///////////////////////////////////////////////////////////////////////////////
// load values into akku1                                                    //
///////////////////////////////////////////////////////////////////////////////
      L    MB10;  // comment
// <- meta.block.fc.body meta.block.network
// ^^^^^^^^^^^^^^^^^^^^^^^^^ meta.block.fc.body meta.block.network
//    ^ keyword.operator.arithmetic.load
//         ^^^^ variable.language.address
//             ^ punctuation.terminator.statement
//                ^^ punctuation.definition.comment.begin
//                ^^^^^^^^^^ comment.line.double-slash
      L    MB[ LD0 ]; // comment
// <- meta.block.fc.body meta.block.network
// ^^^^^^^^^^^^^^^^^^^^^^^^^^^^ meta.block.fc.body meta.block.network
//         ^^^^^^^^^ meta.operand.numeric
//           ^^^^^^^ meta.brackets
//    ^ keyword.operator.arithmetic.load
//         ^^ variable.language.address
//           ^ punctuation.section.brackets.begin
//             ^^^ variable.language.address
//                 ^ punctuation.section.brackets.end
//                  ^ punctuation.terminator.statement
//                    ^^ punctuation.definition.comment.begin
//                    ^^^^^^^^^^ comment.line.double-slash
      L    MW10;  // comment
// <- meta.block.fc.body meta.block.network
// ^^^^^^^^^^^^^^^^^^^^^^^^^ meta.block.fc.body meta.block.network
//    ^ keyword.operator.arithmetic.load
//         ^^^^ variable.language.address
//             ^ punctuation.terminator.statement
//                ^^ punctuation.definition.comment.begin
//                ^^^^^^^^^^ comment.line.double-slash
      L    MW[ LD0 ]; // comment
// <- meta.block.fc.body meta.block.network
// ^^^^^^^^^^^^^^^^^^^^^^^^^^^^ meta.block.fc.body meta.block.network
//         ^^^^^^^^^ meta.operand.numeric
//           ^^^^^^^ meta.brackets
//    ^ keyword.operator.arithmetic.load
//         ^^ variable.language.address
//           ^ punctuation.section.brackets.begin
//             ^^^ variable.language.address
//                 ^ punctuation.section.brackets.end
//                  ^ punctuation.terminator.statement
//                    ^^ punctuation.definition.comment.begin
//                    ^^^^^^^^^^ comment.line.double-slash
      L    MD10;  // comment
// <- meta.block.fc.body meta.block.network
// ^^^^^^^^^^^^^^^^^^^^^^^^^ meta.block.fc.body meta.block.network
//    ^ keyword.operator.arithmetic.load
//         ^^^^ variable.language.address
//             ^ punctuation.terminator.statement
//                ^^ punctuation.definition.comment.begin
//                ^^^^^^^^^^ comment.line.double-slash
      L    MD[ LD0 ]; // comment
// <- meta.block.fc.body meta.block.network
// ^^^^^^^^^^^^^^^^^^^^^^^^^^^^ meta.block.fc.body meta.block.network
//         ^^^^^^^^^ meta.operand.numeric
//           ^^^^^^^ meta.brackets
//    ^ keyword.operator.arithmetic.load
//         ^^ variable.language.address
//           ^ punctuation.section.brackets.begin
//             ^^^ variable.language.address
//                 ^ punctuation.section.brackets.end
//                  ^ punctuation.terminator.statement
//                    ^^ punctuation.definition.comment.begin
//                    ^^^^^^^^^^ comment.line.double-slash
      L    M10.0;  // comment
// <- meta.block.fc.body meta.block.network
// ^^^^^^^^^^^^^^^^^^^^^^^^^^ meta.block.fc.body meta.block.network
//    ^ keyword.operator.arithmetic.load
//         ^^^^^ invalid.illegal
//              ^ punctuation.terminator.statement
//                 ^^ punctuation.definition.comment.begin
//                 ^^^^^^^^^^ comment.line.double-slash
      L    LB10;  // comment
// <- meta.block.fc.body meta.block.network
// ^^^^^^^^^^^^^^^^^^^^^^^^^ meta.block.fc.body meta.block.network
//    ^ keyword.operator.arithmetic.load
//         ^^^^ variable.language.address
//             ^ punctuation.terminator.statement
//                ^^ punctuation.definition.comment.begin
//                ^^^^^^^^^^ comment.line.double-slash
      L    LB[ LD0 ]; // comment
// <- meta.block.fc.body meta.block.network
// ^^^^^^^^^^^^^^^^^^^^^^^^^^^^ meta.block.fc.body meta.block.network
//         ^^^^^^^^^ meta.operand.numeric
//           ^^^^^^^ meta.brackets
//    ^ keyword.operator.arithmetic.load
//         ^^ variable.language.address
//           ^ punctuation.section.brackets.begin
//             ^^^ variable.language.address
//                 ^ punctuation.section.brackets.end
//                  ^ punctuation.terminator.statement
//                    ^^ punctuation.definition.comment.begin
//                    ^^^^^^^^^^ comment.line.double-slash
      L    LW10;  // comment
// <- meta.block.fc.body meta.block.network
// ^^^^^^^^^^^^^^^^^^^^^^^^^ meta.block.fc.body meta.block.network
//    ^ keyword.operator.arithmetic.load
//         ^^^^ variable.language.address
//             ^ punctuation.terminator.statement
//                ^^ punctuation.definition.comment.begin
//                ^^^^^^^^^^ comment.line.double-slash
      L    LW[ LD0 ]; // comment
// <- meta.block.fc.body meta.block.network
// ^^^^^^^^^^^^^^^^^^^^^^^^^^^^ meta.block.fc.body meta.block.network
//         ^^^^^^^^^ meta.operand.numeric
//           ^^^^^^^ meta.brackets
//    ^ keyword.operator.arithmetic.load
//         ^^ variable.language.address
//           ^ punctuation.section.brackets.begin
//             ^^^ variable.language.address
//                 ^ punctuation.section.brackets.end
//                  ^ punctuation.terminator.statement
//                    ^^ punctuation.definition.comment.begin
//                    ^^^^^^^^^^ comment.line.double-slash
      L    LD10;  // comment
// <- meta.block.fc.body meta.block.network
// ^^^^^^^^^^^^^^^^^^^^^^^^^ meta.block.fc.body meta.block.network
//    ^ keyword.operator.arithmetic.load
//         ^^^^ variable.language.address
//             ^ punctuation.terminator.statement
//                ^^ punctuation.definition.comment.begin
//                ^^^^^^^^^^ comment.line.double-slash
      L    LD[ LD0 ]; // comment
// <- meta.block.fc.body meta.block.network
// ^^^^^^^^^^^^^^^^^^^^^^^^^^^^ meta.block.fc.body meta.block.network
//         ^^^^^^^^^ meta.operand.numeric
//           ^^^^^^^ meta.brackets
//    ^ keyword.operator.arithmetic.load
//         ^^ variable.language.address
//           ^ punctuation.section.brackets.begin
//             ^^^ variable.language.address
//                 ^ punctuation.section.brackets.end
//                  ^ punctuation.terminator.statement
//                    ^^ punctuation.definition.comment.begin
//                    ^^^^^^^^^^ comment.line.double-slash
      L    L10.0;  // comment
// <- meta.block.fc.body meta.block.network
// ^^^^^^^^^^^^^^^^^^^^^^^^^^ meta.block.fc.body meta.block.network
//    ^ keyword.operator.arithmetic.load
//         ^^^^^ invalid.illegal
//              ^ punctuation.terminator.statement
//                 ^^ punctuation.definition.comment.begin
//                 ^^^^^^^^^^ comment.line.double-slash
      L     T 10;  // comment
// <- meta.block.fc.body meta.block.network
// ^^^^^^^^^^^^^^^^^^^^^^^^^^ meta.block.fc.body meta.block.network
//    ^ keyword.operator.arithmetic.load
//          ^^^^ variable.language.timer
//              ^ punctuation.terminator.statement
//                 ^^ punctuation.definition.comment.begin
//                 ^^^^^^^^^^ comment.line.double-slash
      L     T [MW10];  // comment
// <- meta.block.fc.body meta.block.network
// ^^^^^^^^^^^^^^^^^^^^^^^^^^^^^ meta.block.fc.body meta.block.network
//     ^^^^^ meta.operand.numeric - meta.address
//          ^^ meta.operand.numeric meta.address.indirect - meta.brackets
//            ^^^^^^ meta.address.indirect meta.brackets
//                  ^^^^^^^^^^^^^^ - meta.operand
//    ^ keyword.operator.arithmetic.load
//          ^ variable.language.timer
//            ^ punctuation.section.brackets.begin
//             ^^^^ variable.language.address
//                 ^ punctuation.section.brackets.end
//                  ^ punctuation.terminator.statement
//                     ^^ punctuation.definition.comment.begin
//                     ^^^^^^^^^^ comment.line.double-slash
      L     Z 10;  // comment
// <- meta.block.fc.body meta.block.network
// ^^^^^^^^^^^^^^^^^^^^^^^^^^ meta.block.fc.body meta.block.network
//    ^ keyword.operator.arithmetic.load
//          ^^^^ variable.language.counter
//              ^ punctuation.terminator.statement
//                 ^^ punctuation.definition.comment.begin
//                 ^^^^^^^^^^ comment.line.double-slash
      L     Z [MW10];  // comment
// <- meta.block.fc.body meta.block.network
// ^^^^^^^^^^^^^^^^^^^^^^^^^^^^^ meta.block.fc.body meta.block.network
//     ^^^^^ meta.operand.numeric - meta.address
//          ^^ meta.operand.numeric meta.address.indirect - meta.brackets
//            ^^^^^^ meta.address.indirect meta.brackets
//                  ^^^^^^^^^^^^^^ - meta.operand
//    ^ keyword.operator.arithmetic.load
//          ^ variable.language.counter
//            ^ punctuation.section.brackets.begin
//             ^^^^ variable.language.address
//                 ^ punctuation.section.brackets.end
//                  ^ punctuation.terminator.statement
//                     ^^ punctuation.definition.comment.begin
//                     ^^^^^^^^^^ comment.line.double-slash
      L     DBNO;  // comment
// <- meta.block.fc.body meta.block.network
// ^^^^^^^^^^^^^^^^^^^^^^^^^^ meta.block.fc.body meta.block.network
//    ^ keyword.operator.arithmetic.load
//          ^^^^ variable.language
//              ^ punctuation.terminator.statement
//                 ^^ punctuation.definition.comment.begin
//                 ^^^^^^^^^^ comment.line.double-slash
      L     DINO;  // comment
// <- meta.block.fc.body meta.block.network
// ^^^^^^^^^^^^^^^^^^^^^^^^^^ meta.block.fc.body meta.block.network
//    ^ keyword.operator.arithmetic.load
//          ^^^^ variable.language
//              ^ punctuation.terminator.statement
//                 ^^ punctuation.definition.comment.begin
//                 ^^^^^^^^^^ comment.line.double-slash
      L     DBB  140;  // comment
// <- meta.block.fc.body meta.block.network
// ^^^^^^^^^^^^^^^^^^^^^^^^^^^^^^ meta.block.fc.body meta.block.network
//    ^ keyword.operator.arithmetic.load
//          ^^^^^^^^ variable.language.address
//                  ^ punctuation.terminator.statement
//                     ^^ punctuation.definition.comment.begin
//                     ^^^^^^^^^^ comment.line.double-slash
      L     DBW  140;  // comment
// <- meta.block.fc.body meta.block.network
// ^^^^^^^^^^^^^^^^^^^^^^^^^^^^^^ meta.block.fc.body meta.block.network
//    ^ keyword.operator.arithmetic.load
//          ^^^^^^^^ variable.language.address
//                  ^ punctuation.terminator.statement
//                     ^^ punctuation.definition.comment.begin
//                     ^^^^^^^^^^ comment.line.double-slash
      L     DBD  140;  // comment
// <- meta.block.fc.body meta.block.network
// ^^^^^^^^^^^^^^^^^^^^^^^^^^^^^^ meta.block.fc.body meta.block.network
//    ^ keyword.operator.arithmetic.load
//          ^^^^^^^^ variable.language.address
//                  ^ punctuation.terminator.statement
//                     ^^ punctuation.definition.comment.begin
//                     ^^^^^^^^^^ comment.line.double-slash
      L     DIB  140;  // comment
// <- meta.block.fc.body meta.block.network
// ^^^^^^^^^^^^^^^^^^^^^^^^^^^^^^ meta.block.fc.body meta.block.network
//    ^ keyword.operator.arithmetic.load
//          ^^^^^^^^ variable.language.address
//                  ^ punctuation.terminator.statement
//                     ^^ punctuation.definition.comment.begin
//                     ^^^^^^^^^^ comment.line.double-slash
      L     DIW  140;  // comment
// <- meta.block.fc.body meta.block.network
// ^^^^^^^^^^^^^^^^^^^^^^^^^^^^^^ meta.block.fc.body meta.block.network
//    ^ keyword.operator.arithmetic.load
//          ^^^^^^^^ variable.language.address
//                  ^ punctuation.terminator.statement
//                     ^^ punctuation.definition.comment.begin
//                     ^^^^^^^^^^ comment.line.double-slash
      L     DID  140;  // comment
// <- meta.block.fc.body meta.block.network
// ^^^^^^^^^^^^^^^^^^^^^^^^^^^^^^ meta.block.fc.body meta.block.network
//    ^ keyword.operator.arithmetic.load
//          ^^^^^^^^ variable.language.address
//                  ^ punctuation.terminator.statement
//                     ^^ punctuation.definition.comment.begin
//                     ^^^^^^^^^^ comment.line.double-slash
      L    DB200.DBB20;  // comment
// <- meta.block.fc.body meta.block.network
// ^^^^^^^^^^^^^^^^^^^^^^^^^^^^^^^^ meta.block.fc.body meta.block.network
//    ^ keyword.operator.arithmetic.load
//         ^^^^^ variable.language.db
//              ^ punctuation.accessor.dot
//               ^^^^^ variable.language.address
//                    ^ punctuation.terminator.statement
//                       ^^ punctuation.definition.comment.begin
//                       ^^^^^^^^^^ comment.line.double-slash
      L    DB200.DBW20;  // comment
// <- meta.block.fc.body meta.block.network
// ^^^^^^^^^^^^^^^^^^^^^^^^^^^^^^^^ meta.block.fc.body meta.block.network
//    ^ keyword.operator.arithmetic.load
//         ^^^^^ variable.language.db
//              ^ punctuation.accessor.dot
//               ^^^^^ variable.language.address
//                    ^ punctuation.terminator.statement
//                       ^^ punctuation.definition.comment.begin
//                       ^^^^^^^^^^ comment.line.double-slash
      L    DB200.DBD20;  // comment
// <- meta.block.fc.body meta.block.network
// ^^^^^^^^^^^^^^^^^^^^^^^^^^^^^^^^ meta.block.fc.body meta.block.network
//    ^ keyword.operator.arithmetic.load
//         ^^^^^ variable.language.db
//              ^ punctuation.accessor.dot
//               ^^^^^ variable.language.address
//                    ^ punctuation.terminator.statement
//                       ^^ punctuation.definition.comment.begin
//                       ^^^^^^^^^^ comment.line.double-slash
      L    DB200.DBX20.0;  // comment
// <- meta.block.fc.body meta.block.network
// ^^^^^^^^^^^^^^^^^^^^^^^^^^^^^^^^^^ meta.block.fc.body meta.block.network
//    ^ keyword.operator.arithmetic.load
//         ^^^^^^^^^^^^^ invalid.illegal
//                      ^ punctuation.terminator.statement
//                         ^^ punctuation.definition.comment.begin
//                         ^^^^^^^^^^ comment.line.double-slash
      L    "datablock".struct[ 4 ].value;  // comment
// <- meta.block.fc.body meta.block.network
// ^^^^^^^^^^^^^^^^^^^^^^^^^^^^^^^^^^^^^^^^^^^^^ meta.block.fc.body meta.block.network
//         ^^^^^^^^^^^^^^^^^^^^^^^^^^^^^ meta.path
//    ^ keyword.operator.arithmetic.load
//         ^ punctuation.definition.variable.begin
//         ^^^^^^^^^^^ variable.namespace
//                   ^ punctuation.definition.variable.end
//                    ^ punctuation.accessor.dot
//                     ^^^^^^ variable.namespace
//                           ^ punctuation.section.brackets.begin
//                           ^^^^^ meta.brackets
//                             ^ meta.number.integer constant.numeric.value
//                               ^ punctuation.section.brackets.end
//                                ^ punctuation.accessor.dot
//                                 ^^^^^ variable.other.member
//                                      ^ punctuation.terminator.statement
//                                         ^^ punctuation.definition.comment.begin
//                                         ^^^^^^^^^^ comment.line.double-slash
      L    "datablock".struct.value;  // comment
// <- meta.block.fc.body meta.block.network
// ^^^^^^^^^^^^^^^^^^^^^^^^^^^^^^^^^^^^^^^^^^^^^ meta.block.fc.body meta.block.network
//         ^^^^^^^^^^^^^^^^^^^^^^^^ meta.path
//    ^ keyword.operator.arithmetic.load
//         ^ punctuation.definition.variable.begin
//         ^^^^^^^^^^^ variable.namespace
//                   ^ punctuation.definition.variable.end
//                    ^ punctuation.accessor.dot
//                     ^^^^^^ variable.namespace
//                           ^ punctuation.accessor.dot
//                            ^^^^^ variable.other.member
//                                 ^ punctuation.terminator.statement
//                                    ^^ punctuation.definition.comment.begin
//                                    ^^^^^^^^^^ comment.line.double-slash
      L    #local[1].array[0].value[ 10 ];  // comment
// <- meta.block.fc.body meta.block.network
// ^^^^^^^^^^^^^^^^^^^^^^^^^^^^^^^^^^^^^^^^^^^^^^ meta.block.fc.body meta.block.network
//    ^ keyword.operator.arithmetic.load
//         ^ punctuation.definition.variable
//         ^^^^^^ variable.namespace
//               ^ punctuation.section.brackets.begin
//               ^^^ meta.brackets
//                ^ meta.number.integer constant.numeric.value
//                 ^ punctuation.section.brackets.end
//                  ^ punctuation.accessor.dot
//                   ^^^^^ variable.namespace
//                        ^ punctuation.section.brackets.begin
//                        ^^^ meta.brackets
//                         ^ meta.number.integer constant.numeric.value
//                          ^ punctuation.section.brackets.end
//                           ^ punctuation.accessor.dot
//                            ^^^^^ variable.other.member
//                                 ^ punctuation.section.brackets.begin
//                                 ^^^^^^ meta.brackets
//                                   ^^ meta.number.integer constant.numeric.value
//                                      ^ punctuation.section.brackets.end
//                                       ^ punctuation.terminator.statement
//                                          ^^ punctuation.definition.comment.begin
//                                          ^^^^^^^^^^ comment.line.double-slash
      L    myNamedValueType#value; // TIA only
//^^^^^^^^^^^^^^^^^^^^^^^^^^^^^^^^ meta.block.fc.body.plc meta.block.network.plc
//    ^ keyword.operator.arithmetic.load.plc
//     ^^^^^^^^^^^^^^^^^^^^^^^^^^ meta.operand.numeric.plc
//         ^^^^^^^^^^^^^^^^ storage.type.enum.plc
//                         ^ punctuation.accessor.plc
//                          ^^^^^ constant.other.enum.plc
//                               ^ punctuation.terminator.statement.plc
      L    "Fancy Named Value Type"#"fancy value"; // TIA only
//^^^^^^^^^^^^^^^^^^^^^^^^^^^^^^^^^^^^^^^^^^^^^^^^ meta.block.fc.body.plc meta.block.network.plc
//    ^ keyword.operator.arithmetic.load.plc
//     ^^^^^^^^^^^^^^^^^^^^^^^^^^^^^^^^^^^^^^^^^^ meta.operand.numeric.plc
//         ^^^^^^^^^^^^^^^^^^^^^^^^ storage.type.enum.plc
//         ^ punctuation.definition.constant.begin.plc
//                                ^ punctuation.definition.constant.end.plc
//                                 ^ punctuation.accessor.plc
//                                  ^^^^^^^^^^^^^ constant.other.enum.plc
//                                  ^ punctuation.definition.constant.begin.plc
//                                              ^ punctuation.definition.constant.end.plc
//                                               ^ punctuation.terminator.statement.plc
      L    P# P0.0; // comment
// <- meta.block.fc.body meta.block.network
// ^^^^^^^^^^^^^^^^^^^^^^^^^^^^^ meta.block.fc.body meta.block.network
//    ^ keyword.operator.arithmetic.load
//         ^^^^^^^ constant.language.pointer
//         ^ storage.type.pointer
//          ^ punctuation.separator.type
//              ^ punctuation.separator.decimal
//                ^ punctuation.terminator.statement
//                  ^^ punctuation.definition.comment.begin
//                  ^^^^^^^^^^ comment.line.double-slash
      L    P##local;  // comment
// <- meta.block.fc.body meta.block.network
// ^^^^^^^^^^^^^^^^^^^^^^^^^^^^^ meta.block.fc.body meta.block.network
//    ^ keyword.operator.arithmetic.load
//         ^ storage.type.pointer
//          ^ punctuation.separator.type
//           ^ punctuation.definition.variable
//            ^^^^^ variable.other.local
//                 ^ punctuation.terminator.statement
//                    ^^ punctuation.definition.comment.begin
//                    ^^^^^^^^^^ comment.line.double-slash
      L    P#120.4;  // comment
// <- meta.block.fc.body meta.block.network
// ^^^^^^^^^^^^^^^^^^^^^^^^^^^^^ meta.block.fc.body meta.block.network
//    ^ keyword.operator.arithmetic.load
//         ^^^^^^^ constant.language.pointer
//         ^ storage.type.pointer
//          ^ punctuation.separator.type
//                ^ punctuation.terminator.statement
//                   ^^ punctuation.definition.comment.begin
//                   ^^^^^^^^^^ comment.line.double-slash
      L    P#DBX120.4;  // comment
// <- meta.block.fc.body meta.block.network
// ^^^^^^^^^^^^^^^^^^^^^^^^^^^^^^^ meta.block.fc.body meta.block.network
//    ^ keyword.operator.arithmetic.load
//         ^^^^^^^^^^ constant.language.pointer
//         ^ storage.type.pointer
//          ^ punctuation.separator.type
//                 ^ punctuation.separator.decimal
//                   ^ punctuation.terminator.statement
//                      ^^ punctuation.definition.comment.begin
//                      ^^^^^^^^^^ comment.line.double-slash
      L    P#DB2.DBX120.4;  // comment
// <- meta.block.fc.body meta.block.network
// ^^^^^^^^^^^^^^^^^^^^^^^^^^^^^^^^^^^^ meta.block.fc.body meta.block.network
//    ^ keyword.operator.arithmetic.load
//         ^^^^^^^^^^^^^^ constant.language.pointer
//         ^ storage.type.pointer
//          ^ punctuation.separator.type
//              ^ punctuation.accessor.dot
//                     ^ punctuation.separator.decimal
//                       ^ punctuation.terminator.statement
//                          ^^ punctuation.definition.comment.begin
//                          ^^^^^^^^^^ comment.line.double-slash
      L    2#0000_0000_0000_0000_0000_0000_0000_0000 ;
// <- meta.block.fc.body meta.block.network
// ^^^^^^^^^^^^^^^^^^^^^^^^^^^^^^^^^^^^^^^^^^^^^^^^^^^^ meta.block.fc.body meta.block.network
//    ^ keyword.operator.arithmetic.load
//         ^^^^^^^^^^^^^^^^^^^^^^^^^^^^^^^^^^^^^^^^^ meta.number.integer.binary
//         ^ constant.numeric.base - punctuation
//          ^ constant.numeric.base punctuation.separator.base
//           ^^^^^^^^^^^^^^^^^^^^^^^^^^^^^^^^^^^^^^^ constant.numeric.value
//               ^ punctuation.separator.digits
//                    ^ punctuation.separator.digits
//                         ^ punctuation.separator.digits
//                              ^ punctuation.separator.digits
//                                   ^ punctuation.separator.digits
//                                        ^ punctuation.separator.digits
//                                             ^ punctuation.separator.digits
//                                                  ^ - invalid
//                                                   ^ punctuation.terminator.statement
//                                                    ^ - invalid
      L    2#1111_1111_1111_1111_1111_1111_1111_1111 ;
// <- meta.block.fc.body meta.block.network
// <- meta.block.fc.body meta.block.network
// ^^^^^^^^^^^^^^^^^^^^^^^^^^^^^^^^^^^^^^^^^^^^^^^^^^^^ meta.block.fc.body meta.block.network
//    ^ keyword.operator.arithmetic.load
//         ^^^^^^^^^^^^^^^^^^^^^^^^^^^^^^^^^^^^^^^^^ meta.number.integer.binary
//         ^ constant.numeric.base - punctuation
//          ^ constant.numeric.base punctuation.separator.base
//           ^^^^^^^^^^^^^^^^^^^^^^^^^^^^^^^^^^^^^^^ constant.numeric.value
//               ^ punctuation.separator.digits
//                    ^ punctuation.separator.digits
//                         ^ punctuation.separator.digits
//                              ^ punctuation.separator.digits
//                                   ^ punctuation.separator.digits
//                                        ^ punctuation.separator.digits
//                                             ^ punctuation.separator.digits
//                                                  ^ - invalid
//                                                   ^ punctuation.terminator.statement
//                                                    ^ - invalid
      L    2#1121_1111_1A11_1111_111_11011_1111_1111 ;
// <- meta.block.fc.body meta.block.network
// ^^^^^^^^^^^^^^^^^^^^^^^^^^^^^^^^^^^^^^^^^^^^^^^^^^^^ meta.block.fc.body meta.block.network
//    ^ keyword.operator.arithmetic.load
//         ^^^^^^^^^^^^^^^^^^^^^^^^^^^^^^^^^^^^^^^^^ meta.number.integer.binary
//         ^ constant.numeric.base - punctuation
//          ^ constant.numeric.base punctuation.separator.base
//           ^^^^^^^^^^^^^^^^^^^^^^^^^^^^^^^^^^^^^^^ constant.numeric.value
//             ^ invalid.illegal.digits
//               ^ punctuation.separator.digits
//                    ^ punctuation.separator.digits
//                      ^ invalid.illegal.digits
//                         ^ punctuation.separator.digits
//                              ^ punctuation.separator.digits
//                                  ^ punctuation.separator.digits
//                                        ^ punctuation.separator.digits
//                                             ^ punctuation.separator.digits
//                                                  ^ - invalid
//                                                   ^ punctuation.terminator.statement
//                                                    ^ - invalid
      L    B#16#0 ;
// <- meta.block.fc.body meta.block.network
// ^^^^^^^^^^^^^^^^^ meta.block.fc.body meta.block.network
//    ^ keyword.operator.arithmetic.load
//         ^^^^^^ meta.number.integer.hexadecimal
//         ^ storage.type.integer
//          ^ punctuation.separator.type
//           ^^ constant.numeric.base - punctuation
//             ^ constant.numeric.base punctuation.separator.base
//              ^ constant.numeric.value
//               ^ - invalid
//                ^ punctuation.terminator.statement
//                 ^ - invalid
      L    byte#16#0 ;
// <- meta.block.fc.body meta.block.network
// ^^^^^^^^^^^^^^^^^^^^ meta.block.fc.body meta.block.network
//    ^ keyword.operator.arithmetic.load
//         ^^^^^^^^^ meta.number.integer.hexadecimal
//         ^^^^ storage.type.integer
//             ^ punctuation.separator.type
//              ^^ constant.numeric.base - punctuation
//                ^ constant.numeric.base punctuation.separator.base
//                 ^ constant.numeric.value
//                  ^ - invalid
//                   ^ punctuation.terminator.statement
//                    ^ - invalid
      L    W#16#0 ;
// <- meta.block.fc.body meta.block.network
// ^^^^^^^^^^^^^^^^^ meta.block.fc.body meta.block.network
//    ^ keyword.operator.arithmetic.load
//         ^^^^^^ meta.number.integer.hexadecimal
//         ^ storage.type.integer
//          ^ punctuation.separator.type
//           ^^ constant.numeric.base - punctuation
//             ^ constant.numeric.base punctuation.separator.base
//              ^ constant.numeric.value
//               ^ - invalid
//                ^ punctuation.terminator.statement
//                 ^ - invalid
      L    word#16#0 ;
// <- meta.block.fc.body meta.block.network
// ^^^^^^^^^^^^^^^^^^^^ meta.block.fc.body meta.block.network
//    ^ keyword.operator.arithmetic.load
//         ^^^^^^^^^ meta.number.integer.hexadecimal
//         ^^^^ storage.type.integer
//             ^ punctuation.separator.type
//              ^^ constant.numeric.base - punctuation
//                ^ constant.numeric.base punctuation.separator.base
//                 ^ constant.numeric.value
//                  ^ - invalid
//                   ^ punctuation.terminator.statement
//                    ^ - invalid
      L    DW#16#0 ;
// <- meta.block.fc.body meta.block.network
// ^^^^^^^^^^^^^^^^^ meta.block.fc.body meta.block.network
//    ^ keyword.operator.arithmetic.load
//         ^^^^^^^ meta.number.integer.hexadecimal
//         ^^ storage.type.integer
//           ^ punctuation.separator.type
//            ^^ constant.numeric.base - punctuation
//              ^ constant.numeric.base punctuation.separator.base
//               ^ constant.numeric.value
//                ^ - invalid
//                 ^ punctuation.terminator.statement
//                  ^ - invalid
      L    dword#16#0 ;
// <- meta.block.fc.body meta.block.network
// ^^^^^^^^^^^^^^^^^^^^^ meta.block.fc.body meta.block.network
//    ^ keyword.operator.arithmetic.load
//         ^^^^^^^^^ meta.number.integer.hexadecimal
//         ^^^^^ storage.type.integer
//              ^ punctuation.separator.type
//               ^^ constant.numeric.base - punctuation
//                 ^ constant.numeric.base punctuation.separator.base
//                  ^ constant.numeric.value
//                   ^ - invalid
//                    ^ punctuation.terminator.statement
//                     ^ - invalid
      L    16 ;
// <- meta.block.fc.body meta.block.network
// ^^^^^^^^^^^^^^^ meta.block.fc.body meta.block.network
//    ^ keyword.operator.arithmetic.load
//         ^^ meta.number.integer.decimal
//         ^^ constant.numeric.value
//           ^ - invalid
//            ^ punctuation.terminator.statement
//             ^ - invalid
      L    -16 ;
// <- meta.block.fc.body meta.block.network
// ^^^^^^^^^^^^^^^ meta.block.fc.body meta.block.network
//    ^ keyword.operator.arithmetic.load
//         ^^^ meta.number.integer.decimal
//         ^ keyword.operator.arithmetic - constant.numeric.value
//          ^^ constant.numeric.value - keyword.operator
//            ^ - invalid
//             ^ punctuation.terminator.statement
//              ^ - invalid
      L    L#16 ;
// <- meta.block.fc.body meta.block.network
// ^^^^^^^^^^^^^^^ meta.block.fc.body meta.block.network
//    ^ keyword.operator.arithmetic.load
//         ^^^^ meta.number.integer.decimal
//         ^ storage.type.integer
//          ^ punctuation.separator.type
//           ^^ constant.numeric.value
//             ^ - invalid
//              ^ punctuation.terminator.statement
//               ^ - invalid
      L    L#-16 ;
// <- meta.block.fc.body meta.block.network
// ^^^^^^^^^^^^^^^ meta.block.fc.body meta.block.network
//    ^ keyword.operator.arithmetic.load
//         ^^^^^ meta.number.integer.decimal
//         ^ storage.type.integer
//          ^ punctuation.separator.type
//           ^ keyword.operator.arithmetic - constant.numeric.value
//            ^^ constant.numeric.value - keyword.operator
//              ^ - invalid
//               ^ punctuation.terminator.statement
//                ^ - invalid
      L    2.0323e+002 ;
// <- meta.block.fc.body meta.block.network
// ^^^^^^^^^^^^^^^^^^^^^^ meta.block.fc.body meta.block.network
//    ^ keyword.operator.arithmetic.load
//         ^^^^^^^^^^^ meta.number.float.decimal constant.numeric.value
//          ^ punctuation.separator.decimal
//                    ^ - invalid
//                     ^ punctuation.terminator.statement
//                      ^ - invalid
      L    -2.0323e-002 ;
// <- meta.block.fc.body meta.block.network
// ^^^^^^^^^^^^^^^^^^^^^^ meta.block.fc.body meta.block.network
//    ^ keyword.operator.arithmetic.load
//         ^^^^^^^^^^^ meta.number.float.decimal
//         ^ keyword.operator.arithmetic - constant.numeric.value
//          ^^^^^^^^^^^ constant.numeric.value - keyword.operator
//           ^ punctuation.separator.decimal
//                     ^ - invalid
//                      ^ punctuation.terminator.statement
//                       ^ - invalid
      L    C#200 ;
// <- meta.block.fc.body meta.block.network
// ^^^^^^^^^^^^^^^^ meta.block.fc.body meta.block.network
//    ^ keyword.operator.arithmetic.load
//         ^^^^^ meta.number.counter.s5
//         ^ storage.type.counter
//          ^ punctuation.separator.type
//           ^^^ constant.numeric.value
//              ^ - invalid
//               ^ punctuation.terminator.statement
//                ^ - invalid
      L     S5T#50MS ;
// <- meta.block.fc.body meta.block.network
// ^^^^^^^^^^^^^^^^^^^ meta.block.fc.body meta.block.network
//    ^ keyword.operator.arithmetic.load
//          ^^^^^^^^ meta.number.time.s5
//          ^^^ storage.type.time
//             ^ punctuation.separator.type
//              ^^ constant.numeric.value.millisecond
//                ^^ constant.numeric.suffix
//                  ^ - invalid
//                   ^ punctuation.terminator.statement
//                    ^ - invalid
      L     S5T#50S ;
// <- meta.block.fc.body meta.block.network
// ^^^^^^^^^^^^^^^^^^ meta.block.fc.body meta.block.network
//    ^ keyword.operator.arithmetic.load
//          ^^^^^^^ meta.number.time.s5
//          ^^^ storage.type.time
//             ^ punctuation.separator.type
//              ^^ constant.numeric.value.second
//                ^ constant.numeric.suffix
//                 ^ - invalid
//                  ^ punctuation.terminator.statement
//                   ^ - invalid
      L     S5T#50M ; //Lade 3000s Sekunden
// <- meta.block.fc.body meta.block.network
// ^^^^^^^^^^^^^^^^^^ meta.block.fc.body meta.block.network
//    ^ keyword.operator.arithmetic.load
//          ^^^^^^^ meta.number.time.s5
//          ^^^ storage.type.time
//             ^ punctuation.separator.type
//              ^^ constant.numeric.value.minute
//                ^ constant.numeric.suffix
//                 ^ - invalid
//                  ^ punctuation.terminator.statement
//                   ^ - invalid
//                    ^^^^^^^^^^^^^^^^^^^^^ comment.line
      L     S5T#1H ;
// <- meta.block.fc.body meta.block.network
// ^^^^^^^^^^^^^^^^^ meta.block.fc.body meta.block.network
//    ^ keyword.operator.arithmetic.load
//          ^^^^^^ meta.number.time.s5
//          ^^^ storage.type.time
//             ^ punctuation.separator.type
//              ^ constant.numeric.value.hour
//               ^ constant.numeric.suffix
//                ^ - invalid
//                 ^ punctuation.terminator.statement
//                  ^ - invalid
      L    S5T#2H_30M_58S_200MS ;
// <- meta.block.fc.body meta.block.network
// ^^^^^^^^^^^^^^^^^^^^^^^^^^^^^^^ meta.block.fc.body meta.block.network
//    ^ keyword.operator.arithmetic.load
//         ^^^^^^^^^^^^^^^^^^^^ meta.number.time.s5
//         ^^^ storage.type.time
//            ^ punctuation.separator.type
//             ^ constant.numeric.value.hour
//              ^ constant.numeric.suffix
//               ^ punctuation.separator.time
//                ^^ constant.numeric.value.minute
//                  ^ constant.numeric.suffix
//                   ^ punctuation.separator.time
//                    ^^ constant.numeric.value.second
//                      ^ constant.numeric.suffix
//                       ^ punctuation.separator.time
//                        ^^^ constant.numeric.value.millisecond
//                           ^^ constant.numeric.suffix
//                             ^ - invalid
//                              ^ punctuation.terminator.statement
//                               ^ - invalid
      L    S5T#2H_70M_58S_200MS ;
// <- meta.block.fc.body meta.block.network
// ^^^^^^^^^^^^^^^^^^^^^^^^^^^^^^^ meta.block.fc.body meta.block.network
//    ^ keyword.operator.arithmetic.load
//         ^^^^^^^^^^^^^^^^^^^^ meta.number.time.s5
//         ^^^ storage.type.time
//            ^ punctuation.separator.type
//             ^ constant.numeric.value.hour
//              ^ constant.numeric.suffix
//               ^ punctuation.separator.time
//                ^^ constant.numeric.value.minute.plc
//                  ^ constant.numeric.suffix.minute.plc
//                   ^ punctuation.separator.time
//                    ^^ constant.numeric.value.second
//                      ^ constant.numeric.suffix
//                       ^ punctuation.separator.time
//                        ^^^ constant.numeric.value.millisecond
//                           ^^ constant.numeric.suffix
//                             ^ - invalid
//                              ^ punctuation.terminator.statement
//                               ^ - invalid
      L     T#50MS ;
// <- meta.block.fc.body meta.block.network
// ^^^^^^^^^^^^^^^^^ meta.block.fc.body meta.block.network
//    ^ keyword.operator.arithmetic.load
//          ^^^^^^ meta.number.time.iec
//          ^ storage.type.time
//           ^ punctuation.separator.type
//            ^^ constant.numeric.value.millisecond
//              ^^ constant.numeric.suffix
//                ^ - invalid
//                 ^ punctuation.terminator.statement
//                  ^ - invalid
      L     T#50S ;
// <- meta.block.fc.body meta.block.network
// ^^^^^^^^^^^^^^^^^ meta.block.fc.body meta.block.network
//    ^ keyword.operator.arithmetic.load
//          ^^^^^ meta.number.time.iec
//          ^ storage.type.time
//           ^ punctuation.separator.type
//            ^^ constant.numeric.value.second
//              ^ constant.numeric.suffix
//               ^ - invalid
//                ^ punctuation.terminator.statement
//                 ^ - invalid
      L     T#50M ;
// <- meta.block.fc.body meta.block.network
// ^^^^^^^^^^^^^^^^^ meta.block.fc.body meta.block.network
//    ^ keyword.operator.arithmetic.load
//          ^^^^^ meta.number.time.iec
//          ^ storage.type.time
//           ^ punctuation.separator.type
//            ^^ constant.numeric.value.minute
//              ^ constant.numeric.suffix
//               ^ - invalid
//                ^ punctuation.terminator.statement
//                 ^ - invalid
      L     T#1H ;
// <- meta.block.fc.body meta.block.network
// ^^^^^^^^^^^^^^^^ meta.block.fc.body meta.block.network
//    ^ keyword.operator.arithmetic.load
//          ^^^^ meta.number.time.iec
//          ^ storage.type.time
//           ^ punctuation.separator.type
//            ^ constant.numeric.value.hour
//             ^ constant.numeric.suffix
//              ^ - invalid
//               ^ punctuation.terminator.statement
//                ^ - invalid
      L     T#2D ;
// <- meta.block.fc.body meta.block.network
// ^^^^^^^^^^^^^^^^ meta.block.fc.body meta.block.network
//    ^ keyword.operator.arithmetic.load
//          ^^^^ meta.number.time.iec
//          ^ storage.type.time
//           ^ punctuation.separator.type
//            ^ constant.numeric.value.day
//             ^ constant.numeric.suffix
//              ^ - invalid
//               ^ punctuation.terminator.statement
//                ^ - invalid
      L    T#24D_23H_59M_59S_999MS ;
// <- meta.block.fc.body meta.block.network
// ^^^^^^^^^^^^^^^^^^^^^^^^^^^^^^^^^^ meta.block.fc.body meta.block.network
//    ^ keyword.operator.arithmetic.load
//         ^^^^^^^^^^^^^^^^^^^^^^^ meta.number.time.iec
//         ^ storage.type.time
//          ^ punctuation.separator.type
//           ^^ constant.numeric.value.day
//             ^ constant.numeric.suffix
//              ^ punctuation.separator.time
//               ^^ constant.numeric.value.hour
//                 ^ constant.numeric.suffix
//                  ^ punctuation.separator.time
//                   ^^ constant.numeric.value.minute
//                     ^ constant.numeric.suffix
//                      ^ punctuation.separator.time
//                       ^^ constant.numeric.value.second
//                         ^ constant.numeric.suffix
//                          ^ punctuation.separator.time
//                           ^^^ constant.numeric.value.millisecond
//                              ^^ constant.numeric.suffix
//                                ^ - invalid
//                                 ^ punctuation.terminator.statement
//                                  ^ - invalid
      L    T#25D_23H_69M_59S_999MS ;
// <- meta.block.fc.body meta.block.network
// ^^^^^^^^^^^^^^^^^^^^^^^^^^^^^^^^^^ meta.block.fc.body meta.block.network
//    ^ keyword.operator.arithmetic.load
//         ^^^^^^^^^^^^^^^^^^^^^^^ meta.number.time.iec
//         ^ storage.type.time
//          ^ punctuation.separator.type
//           ^^^ invalid.illegal.time.day
//              ^ punctuation.separator.time
//               ^^ constant.numeric.value.hour
//                 ^ constant.numeric.suffix
//                  ^ punctuation.separator.time
//                   ^^ constant.numeric.value.minute.plc
//                     ^ constant.numeric.suffix.minute.plc
//                      ^ punctuation.separator.time
//                       ^^ constant.numeric.value.second
//                         ^ constant.numeric.suffix
//                          ^ punctuation.separator.time
//                           ^^^ constant.numeric.value.millisecond
//                              ^^ constant.numeric.suffix
//                                ^ - invalid
//                                 ^ punctuation.terminator.statement
//                                  ^ - invalid
      L    t#25d_23h_69m_59s_999ms ;
// <- meta.block.fc.body meta.block.network
// ^^^^^^^^^^^^^^^^^^^^^^^^^^^^^^^^^^ meta.block.fc.body meta.block.network
//    ^ keyword.operator.arithmetic.load
//         ^^^^^^^^^^^^^^^^^^^^^^^ meta.number.time.iec
//         ^ storage.type.time
//          ^ punctuation.separator.type
//           ^^^ invalid.illegal.time.day
//              ^ punctuation.separator.time
//               ^^ constant.numeric.value.hour
//                 ^ constant.numeric.suffix
//                  ^ punctuation.separator.time
//                   ^^ constant.numeric.value.minute.plc
//                     ^ constant.numeric.suffix.minute.plc
//                      ^ punctuation.separator.time
//                       ^^ constant.numeric.value.second
//                         ^ constant.numeric.suffix
//                          ^ punctuation.separator.time
//                           ^^^ constant.numeric.value.millisecond
//                              ^^ constant.numeric.suffix
//                                ^ - invalid
//                                 ^ punctuation.terminator.statement
//                                  ^ - invalid
      L    T#24D_23M_59M_20H_999MS ;
// <- meta.block.fc.body meta.block.network
// ^^^^^^^^^^^^^^^^^^^^^^^^^^^^^^^^^^ meta.block.fc.body meta.block.network
//    ^ keyword.operator.arithmetic.load
//         ^^^^^^^^^^^^^^^^^^^^^^^ meta.number.time.iec
//         ^ storage.type.time
//          ^ punctuation.separator.type
//           ^^ constant.numeric.value.day
//             ^ constant.numeric.suffix
//              ^ punctuation.separator.time
//               ^^^ invalid.illegal.time.hour
//                  ^ punctuation.separator.time
//                   ^^ constant.numeric.value.minute
//                     ^ constant.numeric.suffix
//                      ^ punctuation.separator.time
//                       ^^^ invalid.illegal.time.second
//                          ^ punctuation.separator.time
//                           ^^^ constant.numeric.value.millisecond
//                              ^^ constant.numeric.suffix
//                                ^ - invalid
//                                 ^ punctuation.terminator.statement
//                                  ^ - invalid

      L    LT#999ns LT#-999ns LT#+999ns
//         ^^^^^^^^ meta.number.time.iec.plc
//         ^^ storage.type.time.plc
//           ^ punctuation.separator.type.plc
//            ^^^ constant.numeric.value.nanosecond.plc
//               ^^ constant.numeric.suffix.nanosecond.plc
//                  ^^^^^^^^^ meta.number.time.iec.plc
//                  ^^ storage.type.time.plc
//                    ^ punctuation.separator.type.plc
//                     ^ constant.numeric.value.plc keyword.operator.arithmetic.plc
//                      ^^^ constant.numeric.value.nanosecond.plc
//                         ^^ constant.numeric.suffix.nanosecond.plc
//                            ^^^^^^^^^ meta.number.time.iec.plc
//                            ^^ storage.type.time.plc
//                              ^ punctuation.separator.type.plc
//                               ^ constant.numeric.value.plc keyword.operator.arithmetic.plc
//                                ^^^ constant.numeric.value.nanosecond.plc
//                                   ^^ constant.numeric.suffix.nanosecond.plc

      L    LT#999us LT#-999us LT#+999us
//         ^^^^^^^^ meta.number.time.iec.plc
//         ^^ storage.type.time.plc
//           ^ punctuation.separator.type.plc
//            ^^^ constant.numeric.value.microsecond.plc
//               ^^ constant.numeric.suffix.microsecond.plc
//                  ^^^^^^^^^ meta.number.time.iec.plc
//                  ^^ storage.type.time.plc
//                    ^ punctuation.separator.type.plc
//                     ^ constant.numeric.value.plc keyword.operator.arithmetic.plc
//                      ^^^ constant.numeric.value.microsecond.plc
//                         ^^ constant.numeric.suffix.microsecond.plc
//                            ^^^^^^^^^ meta.number.time.iec.plc
//                            ^^ storage.type.time.plc
//                              ^ punctuation.separator.type.plc
//                               ^ constant.numeric.value.plc keyword.operator.arithmetic.plc
//                                ^^^ constant.numeric.value.microsecond.plc
//                                   ^^ constant.numeric.suffix.microsecond.plc

      L    LT#999ms LT#-999ms LT#+999ms
//         ^^^^^^^^ meta.number.time.iec.plc
//         ^^ storage.type.time.plc
//           ^ punctuation.separator.type.plc
//            ^^^ constant.numeric.value.millisecond.plc
//               ^^ constant.numeric.suffix.millisecond.plc
//                  ^^^^^^^^^ meta.number.time.iec.plc
//                  ^^ storage.type.time.plc
//                    ^ punctuation.separator.type.plc
//                     ^ constant.numeric.value.plc keyword.operator.arithmetic.plc
//                      ^^^ constant.numeric.value.millisecond.plc
//                         ^^ constant.numeric.suffix.millisecond.plc
//                            ^^^^^^^^^ meta.number.time.iec.plc
//                            ^^ storage.type.time.plc
//                              ^ punctuation.separator.type.plc
//                               ^ constant.numeric.value.plc keyword.operator.arithmetic.plc
//                                ^^^ constant.numeric.value.millisecond.plc
//                                   ^^ constant.numeric.suffix.millisecond.plc

      L    LT#-106751d_23h_47m_16s_854ms_775us_808ns
//         ^^^^^^^^^^^^^^^^^^^^^^^^^^^^^^^^^^^^^^^^^ meta.number.time.iec.plc - invalid
//         ^^ storage.type.time.plc
//           ^ punctuation.separator.type.plc
//            ^ constant.numeric.value.plc keyword.operator.arithmetic.plc
//             ^^^^^^ constant.numeric.value.day.plc
//                   ^ constant.numeric.suffix.day.plc
//                    ^ punctuation.separator.time.plc
//                     ^^ constant.numeric.value.hour.plc
//                       ^ constant.numeric.suffix.hour.plc
//                        ^ punctuation.separator.time.plc
//                         ^^ constant.numeric.value.minute.plc
//                           ^ constant.numeric.suffix.minute.plc
//                            ^ punctuation.separator.time.plc
//                             ^^ constant.numeric.value.second.plc
//                               ^ constant.numeric.suffix.second.plc
//                                ^ punctuation.separator.time.plc
//                                 ^^^ constant.numeric.value.millisecond.plc
//                                    ^^ constant.numeric.suffix.millisecond.plc
//                                      ^ punctuation.separator.time.plc
//                                       ^^^ constant.numeric.value.microsecond.plc
//                                          ^^ constant.numeric.suffix.microsecond.plc
//                                            ^ punctuation.separator.time.plc
//                                             ^^^ constant.numeric.value.nanosecond.plc
//                                                ^^ constant.numeric.suffix.nanosecond.plc

      L    LT#+106751d_23h_47m_16s_854ms_775us_807ns
//         ^^^^^^^^^^^^^^^^^^^^^^^^^^^^^^^^^^^^^^^^^ meta.number.time.iec.plc - invalid
//         ^^ storage.type.time.plc
//           ^ punctuation.separator.type.plc
//            ^ constant.numeric.value.plc keyword.operator.arithmetic.plc
//             ^^^^^^ constant.numeric.value.day.plc
//                   ^ constant.numeric.suffix.day.plc
//                    ^ punctuation.separator.time.plc
//                     ^^ constant.numeric.value.hour.plc
//                       ^ constant.numeric.suffix.hour.plc
//                        ^ punctuation.separator.time.plc
//                         ^^ constant.numeric.value.minute.plc
//                           ^ constant.numeric.suffix.minute.plc
//                            ^ punctuation.separator.time.plc
//                             ^^ constant.numeric.value.second.plc
//                               ^ constant.numeric.suffix.second.plc
//                                ^ punctuation.separator.time.plc
//                                 ^^^ constant.numeric.value.millisecond.plc
//                                    ^^ constant.numeric.suffix.millisecond.plc
//                                      ^ punctuation.separator.time.plc
//                                       ^^^ constant.numeric.value.microsecond.plc
//                                          ^^ constant.numeric.suffix.microsecond.plc
//                                            ^ punctuation.separator.time.plc
//                                             ^^^ constant.numeric.value.nanosecond.plc
//                                                ^^ constant.numeric.suffix.nanosecond.plc

      L    LT#+106752d_23h_47m_16s_854ms_775us_807ns
//         ^^^^^^^^^^^^^^^^^^^^^^^^^^^^^^^^^^^^^^^^^ meta.number.time.iec.plc
//         ^^ storage.type.time.plc
//           ^ punctuation.separator.type.plc
//            ^ constant.numeric.value.plc keyword.operator.arithmetic.plc
//             ^^^^^^^ invalid.illegal.time.day.plc
//                    ^ punctuation.separator.time.plc
//                     ^^ constant.numeric.value.hour.plc
//                       ^ constant.numeric.suffix.hour.plc
//                        ^ punctuation.separator.time.plc
//                         ^^ constant.numeric.value.minute.plc
//                           ^ constant.numeric.suffix.minute.plc
//                            ^ punctuation.separator.time.plc
//                             ^^ constant.numeric.value.second.plc
//                               ^ constant.numeric.suffix.second.plc
//                                ^ punctuation.separator.time.plc
//                                 ^^^ constant.numeric.value.millisecond.plc
//                                    ^^ constant.numeric.suffix.millisecond.plc
//                                      ^ punctuation.separator.time.plc
//                                       ^^^ constant.numeric.value.microsecond.plc
//                                          ^^ constant.numeric.suffix.microsecond.plc
//                                            ^ punctuation.separator.time.plc
//                                             ^^^ constant.numeric.value.nanosecond.plc
//                                                ^^ constant.numeric.suffix.nanosecond.plc

      L    DT#1970-01-01-00:00:00 ;
//         ^^^^^^^^^^^^^^^^^^^^^^ meta.number.date-and-time.plc
//         ^^ storage.type.time.plc
//           ^ punctuation.separator.type.plc
//            ^^^^^^^^^^^^^^^^^^^ constant.numeric.value.plc
//                ^ punctuation.separator.date.plc
//                   ^ punctuation.separator.date.plc
//                         ^ punctuation.separator.time.plc
//                            ^ punctuation.separator.time.plc

      L    LDT#1970-01-01-00:00:00 ;
//         ^^^^^^^^^^^^^^^^^^^^^^^ meta.number.date-and-time.plc
//         ^^^ storage.type.time.plc
//            ^ punctuation.separator.type.plc
//             ^^^^^^^^^^^^^^^^^^^ constant.numeric.value.plc
//                 ^ punctuation.separator.date.plc
//                    ^ punctuation.separator.date.plc
//                          ^ punctuation.separator.time.plc
//                             ^ punctuation.separator.time.plc

      L    D#2017-12-30 ;
// <- meta.block.fc.body meta.block.network
// ^^^^^^^^^^^^^^^^^^^^^^^ meta.block.fc.body meta.block.network
//    ^ keyword.operator.arithmetic.load
//         ^^^^^^^^^^^^ meta.number.date
//         ^ storage.type.time
//          ^ punctuation.separator.type
//           ^^^^^^^^^^ constant.numeric.value
//               ^ punctuation.separator.date
//                  ^ punctuation.separator.date
//                     ^ - invalid
//                      ^ punctuation.terminator.statement
//                       ^ - invalid

      L    DATE#2017-12-30 ;
// <- meta.block.fc.body meta.block.network
// ^^^^^^^^^^^^^^^^^^^^^^^^^^ meta.block.fc.body meta.block.network
//    ^ keyword.operator.arithmetic.load
//         ^^^^^^^^^^^^^^^ meta.number.date
//         ^^^^ storage.type.time
//             ^ punctuation.separator.type
//              ^^^^^^^^^^ constant.numeric.value
//                  ^ punctuation.separator.date
//                     ^ punctuation.separator.date
//                        ^ - invalid
//                         ^ punctuation.terminator.statement
//                          ^ - invalid

      L    LDATE#2162-12-30 ;
//         ^^^^^^^^^^^^^^^^ meta.number.date.plc
//         ^^^^^ storage.type.time.plc
//              ^ punctuation.separator.type.plc
//               ^^^^^^^^^^ constant.numeric.value.plc
//                   ^ punctuation.separator.date.plc
//                      ^ punctuation.separator.date.plc
//                         ^ - invalid
//                          ^ punctuation.terminator.statement.plc
//                           ^ - invalid

      L    TOD#23:59:59.999 ;
// <- meta.block.fc.body meta.block.network
// ^^^^^^^^^^^^^^^^^^^^^^^^^^^ meta.block.fc.body meta.block.network
//    ^ keyword.operator.arithmetic.load
//         ^^^^^^^^^^^^^^^^ meta.number.time-of-day
//         ^^^ storage.type.time
//            ^ punctuation.separator.type
//             ^^^^^^^^^^^^ constant.numeric.value
//               ^ punctuation.separator.time
//                  ^ punctuation.separator.time
//                     ^ punctuation.separator.time
//                         ^ - invalid
//                          ^ punctuation.terminator.statement
//                           ^ - invalid

      L    LTOD#23:59:59.999 ;
//         ^^^^^^^^^^^^^^^^^ meta.number.time-of-day.plc
//         ^^^^ storage.type.time.plc
//             ^ punctuation.separator.type.plc
//              ^^^^^^^^^^^^ constant.numeric.value.plc
//                ^ punctuation.separator.time.plc
//                   ^ punctuation.separator.time.plc
//                      ^ punctuation.separator.time.plc
//                          ^ - invalid
//                           ^ punctuation.terminator.statement.plc
//                            ^ - invalid

      L    'A'
//    ^ keyword.operator.arithmetic.load
//         ^^^ meta.string string.quoted.single
//         ^ punctuation.definition.string.begin
//          ^ constant.character.literal
//           ^ punctuation.definition.string.end

///////////////////////////////////////////////////////////////////////////////
// aritmetic operations                                                      //
///////////////////////////////////////////////////////////////////////////////

      +    16 ;
// <- meta.block.fc.body meta.block.network
// ^^^^^^^^^^^^^^^ meta.block.fc.body meta.block.network
//    ^ keyword.operator.arithmetic
//         ^^ meta.number.integer.decimal
//         ^^ constant.numeric.value
//           ^ - invalid
//            ^ punctuation.terminator.statement
//             ^ - invalid
      +    -16 ;
// <- meta.block.fc.body meta.block.network
// ^^^^^^^^^^^^^^^ meta.block.fc.body meta.block.network
//    ^ keyword.operator.arithmetic
//         ^^^ meta.number.integer.decimal
//         ^ keyword.operator.arithmetic - constant.numeric.value
//          ^^ constant.numeric.value - keyword.operator
//            ^ - invalid
//             ^ punctuation.terminator.statement
//              ^ - invalid
      +    L#16 ;
// <- meta.block.fc.body meta.block.network
// ^^^^^^^^^^^^^^^ meta.block.fc.body meta.block.network
//    ^ keyword.operator.arithmetic
//         ^^^^ meta.number.integer.decimal
//         ^ storage.type.integer
//          ^ punctuation.separator.type
//           ^^ constant.numeric.value
//             ^ - invalid
//              ^ punctuation.terminator.statement
//               ^ - invalid
      +    L#-16 ;
// <- meta.block.fc.body meta.block.network
// ^^^^^^^^^^^^^^^ meta.block.fc.body meta.block.network
//    ^ keyword.operator.arithmetic
//         ^^^^^ meta.number.integer.decimal
//         ^ storage.type.integer
//          ^ punctuation.separator.type
//           ^ keyword.operator.arithmetic - constant.numeric.value
//            ^^ constant.numeric.value - keyword.operator
//              ^ - invalid
//               ^ punctuation.terminator.statement
//                ^ - invalid

      +     DINT#10 ;
//^^^^^^^^^^^^^^^^^^^^ meta.block.fc.body.plc meta.block.network.plc
//    ^ keyword.operator.arithmetic.plc
//     ^^^^^^^^^^^^^ meta.operand.constant.numeric.plc
//          ^^^^^^^ meta.number.integer.decimal.plc
//          ^^^^ storage.type.integer.plc
//              ^ punctuation.separator.type.plc
//               ^^ constant.numeric.value.plc
//                 ^ - invalid
//                  ^ punctuation.terminator.statement.plc
//                   ^ - invalid

///////////////////////////////////////////////////////////////////////////////
// function calls                                                            //
///////////////////////////////////////////////////////////////////////////////

      CALL "ALARM_SQ" (
// <- meta.block.fc.body meta.block.network
// ^^^^^^^^^^^^^^^^^^^^ meta.block.fc.body meta.block.network
//    ^^^^ meta.function-call - meta.function-call meta.function-call
//        ^^^^^^^^^^^^ meta.function-call.identifier - meta.function-call meta.function-call
//                    ^ meta.function-call.arguments - meta.function-call meta.function-call
//    ^^^^ keyword.control.call
//         ^ variable.function.global punctuation.definition.variable.begin
//          ^^^^^^^^ variable.function.global - punctuation
//                  ^ variable.function.global punctuation.definition.variable.end
//                    ^ punctuation.section.group.begin
           EN      := L 4.0,
// <- meta.block.fc.body meta.block.network meta.function-call.arguments
// ^^^^^^^^^^^^^^^^^^^^^^^^^^ meta.block.fc.body meta.block.network meta.function-call.arguments
//         ^^ variable.parameter
//                 ^^ keyword.operator.assignment
//                    ^^^^^ variable.language.address
//                         ^ punctuation.separator.sequence
           INTF    := DB 2,
// <- meta.block.fc.body meta.block.network meta.function-call.arguments
// ^^^^^^^^^^^^^^^^^^^^^^^^^^ meta.block.fc.body meta.block.network meta.function-call.arguments
//         ^^^^ variable.parameter
//                 ^^ keyword.operator.assignment
//                    ^^^^ variable.language.db
//                        ^ punctuation.separator.sequence
           TMR     := T 2,
// <- meta.block.fc.body meta.block.network meta.function-call.arguments
// ^^^^^^^^^^^^^^^^^^^^^^^^^^ meta.block.fc.body meta.block.network meta.function-call.arguments
//         ^^^ variable.parameter
//                 ^^ keyword.operator.assignment
//                    ^^^ variable.language.timer
//                       ^ punctuation.separator.sequence
           CNT     := Z 2,
// <- meta.block.fc.body meta.block.network meta.function-call.arguments
// ^^^^^^^^^^^^^^^^^^^^^^^^^^ meta.block.fc.body meta.block.network meta.function-call.arguments
//         ^^^ variable.parameter
//                 ^^ keyword.operator.assignment
//                    ^^^ variable.language.counter
//                       ^ punctuation.separator.sequence
           SIG     := "msgs".A700127,
// <- meta.block.fc.body meta.block.network meta.function-call.arguments
// ^^^^^^^^^^^^^^^^^^^^^^^^^^^^^^^^^^ meta.block.fc.body meta.block.network meta.function-call.arguments
//         ^^^ variable.parameter
//                 ^^ keyword.operator.assignment
//                    ^^^^^^^^^^^^^^ meta.path
//                    ^^^^^^ variable.namespace
//                    ^ punctuation.definition.variable.begin
//                         ^ punctuation.definition.variable.end
//                          ^ punctuation.accessor
//                           ^^^^^^^ variable.other.member
//                                  ^ punctuation.separator.sequence
           ID      := W#16#EEEE,
// <- meta.block.fc.body meta.block.network meta.function-call.arguments
// ^^^^^^^^^^^^^^^^^^^^^^^^^^^^^ meta.block.fc.body meta.block.network meta.function-call.arguments
//         ^^ variable.parameter
//                 ^^ keyword.operator.assignment
//                    ^^^^^^^^^ meta.number.integer.hexadecimal
//                             ^ punctuation.separator.sequence
           EV_ID   := DW#16#AAEDF,
// <- meta.block.fc.body meta.block.network meta.function-call.arguments
// ^^^^^^^^^^^^^^^^^^^^^^^^^^^^^^ meta.block.fc.body meta.block.network meta.function-call.arguments
//         ^^^^^ variable.parameter
//                 ^^ keyword.operator.assignment
//                    ^^^^^^^^^^^ meta.number.integer.hexadecimal
//                               ^ punctuation.separator.sequence
           ANY     := P# DB20.DBX40.0 WORD 10,
// <- meta.block.fc.body meta.block.network meta.function-call.arguments
// ^^^^^^^^^^^^^^^^^^^^^^^^^ meta.block.fc.body meta.block.network meta.function-call.arguments
//                                    ^^^^ storage.type
//         ^^ variable.parameter
//                 ^^ keyword.operator.assignment
//                    ^^^^^^^^^^^^^^^^^^^^^^^ constant.language.any-pointer
//                                           ^ punctuation.separator.sequence
           OTHER   := NULL,
// <- meta.block.fc.body meta.block.network meta.function-call.arguments
// ^^^^^^^^^^^^^^^^^^^^^^^^^ meta.block.fc.body meta.block.network meta.function-call.arguments
//         ^^^^^ variable.parameter
//                 ^^ keyword.operator.assignment
//                    ^^^^ constant.language.null
//                        ^ punctuation.separator.sequence
           SD      := #data,
// <- meta.block.fc.body meta.block.network meta.function-call.arguments
// ^^^^^^^^^^^^^^^^^^^^^^^^^ meta.block.fc.body meta.block.network meta.function-call.arguments
//         ^^ variable.parameter
//                 ^^ keyword.operator.assignment
//                    ^^^^^ variable.other.local
//                    ^ punctuation.definition.variable
//                         ^ punctuation.separator.sequence
           "quoted:=arg" := 'value',
// <- meta.block.fc.body meta.block.network meta.function-call.arguments
// ^^^^^^^^^^^^^^^^^^^^^^^^^^^^^^^^^ meta.block.fc.body meta.block.network meta.function-call.arguments
//         ^^^^^^^^^^^^^ variable.parameter.plc
//         ^ punctuation.definition.variable.begin.plc
//                     ^ punctuation.definition.variable.end.plc
//                       ^^ keyword.operator.assignment.plc
//                          ^^^^^^^ meta.string.plc string.quoted.single.plc

           RET_VAL := MW200);
// <- meta.block.fc.body meta.block.network meta.function-call.arguments
// ^^^^^^^^^^^^^^^^^^^^^^^^^ meta.block.fc.body meta.block.network meta.function-call.arguments
//         ^^^^^^^ variable.parameter
//                 ^^ keyword.operator.assignment
//                    ^^^^^ variable.language.address
//                         ^ punctuation.section.group.end
//                          ^ punctuation.terminator.statement
   CALL #wdgPrgRead
   {time_type := 'Time'}
//^ meta.function-call.identifier.plc
// ^^^^^^^^^^^^^^^^^^^^^ meta.function-call.plc meta.annotation.plc
//                      ^ meta.function-call.plc - meta.annotation

   CALL #wdgPrgRead
   {time_type := 'Time'}
   (  IN := #interface.Platz.PrgReadReq ,
//^ meta.function-call.plc - meta.annotation - meta.group
// ^^^^^^^^^^^^^^^^^^^^^^^^^^^^^^^^^^^^^^^ meta.function-call.arguments.plc meta.group.plc
// ^ punctuation.section.group.begin.plc
//    ^^ variable.parameter.plc
//       ^^ keyword.operator.assignment.plc
   );
//^^ meta.function-call.arguments.plc meta.group.plc
//  ^ - meta.function-call
// ^ punctuation.section.group.end.plc
//  ^ punctuation.terminator.statement.plc

   CALL FC 10 ();
// ^^^^ meta.function-call
//     ^^^^^^^ meta.function-call.identifier
//            ^^ meta.function-call.arguments
// ^^^^ keyword.control.call
//      ^^^^^ variable.function.address
//            ^ punctuation.section.group.begin
//             ^ punctuation.section.group.end

   CALL SFC 10 ();
// ^^^^ meta.function-call
//     ^^^^^^^^ meta.function-call.identifier
//             ^^ meta.function-call.arguments
// ^^^^ keyword.control.call
//      ^^^^^^ variable.function.address
//             ^ punctuation.section.group.begin
//              ^ punctuation.section.group.end

   CALL FB 10, DB 10 ();
// ^^^^ meta.function-call - meta.function-call meta.function-call
//     ^^^^^^ meta.function-call.identifier - meta.function-call meta.function-call
//           ^ meta.function-call - meta.function-call meta.function-call
//            ^^^^^^^ meta.function-call.instance - meta.function-call meta.function-call
//                   ^^ meta.function-call.arguments - meta.function-call meta.function-call
// ^^^^ keyword.control.call
//      ^^^^^ variable.function.address
//           ^ punctuation.separator.sequence
//             ^^^^^ variable.language.db
//                   ^ punctuation.section.group.begin
//                    ^ punctuation.section.group.end

   CALL "Block", "InstDB" ();
// ^^^^ meta.function-call - meta.function-call meta.function-call
//     ^^^^^^^^ meta.function-call.identifier - meta.function-call meta.function-call
//             ^ meta.function-call - meta.function-call meta.function-call
//              ^^^^^^^^^^ meta.function-call.instance - meta.function-call meta.function-call
//                        ^^ meta.function-call.arguments - meta.function-call meta.function-call
// ^^^^ keyword.control.call
//      ^ variable.function.global punctuation.definition.variable.begin
//       ^^^^^ variable.function.global - punctuation
//            ^ variable.function.global punctuation.definition.variable.end
//             ^ punctuation.separator.sequence
//               ^^^^^^^^ variable.other.global
//                        ^ punctuation.section.group.begin
//                         ^ punctuation.section.group.end

   CALL BLKMOV
//^^^^^^^^^^^^ meta.block.fc.body.plc meta.block.network.plc
// ^^^^ meta.function-call.plc keyword.control.call.plc
//     ^^^^^^^ meta.function-call.identifier.plc
//      ^^^^^^ support.function.built-in.plc
   {blk_type := 'Variant'}
//^^^^^^^^^^^^^^^^^^^^^^^^ meta.block.fc.body.plc meta.block.network.plc
//^ meta.function-call.identifier.plc
// ^^^^^^^^^^^^^^^^^^^^^^^ meta.function-call.plc meta.annotation.plc
// ^ punctuation.definition.annotation.begin.plc
//  ^^^^^^^^ variable.annotation.plc
//           ^^ keyword.operator.assignment.plc
//              ^^^^^^^^^ meta.string.plc string.quoted.single.plc
//              ^ punctuation.definition.string.begin.plc
//                      ^ punctuation.definition.string.end.plc
//                       ^ punctuation.definition.annotation.end.plc
   (  SRCBLK                      := "DB1".src ,
//^^^^^^^^^^^^^^^^^^^^^^^^^^^^^^^^^^^^^^^^^^^^^^ meta.block.fc.body.plc meta.block.network.plc
//^ meta.function-call.plc
// ^^^^^^^^^^^^^^^^^^^^^^^^^^^^^^^^^^^^^^^^^^^^^ meta.function-call.arguments.plc meta.group.plc
// ^ punctuation.section.group.begin.plc
//    ^^^^^^ variable.parameter.plc
//                                ^^ keyword.operator.assignment.plc
//                                   ^^^^^^^^^^ meta.path.plc
//                                   ^^^^^ variable.namespace.plc
//                                   ^ punctuation.definition.variable.begin.plc
//                                       ^ punctuation.definition.variable.end.plc
//                                        ^ punctuation.accessor.dot.plc
//                                         ^^^ variable.other.member.plc
//                                             ^ punctuation.separator.sequence.plc
      RET_VAL                     := #STATUS ,
//^^^^^^^^^^^^^^^^^^^^^^^^^^^^^^^^^^^^^^^^^^^^^ meta.block.fc.body.plc meta.block.network.plc meta.function-call.arguments.plc meta.group.plc
//    ^^^^^^^ variable.parameter.plc
//                                ^^ keyword.operator.assignment.plc
//                                   ^^^^^^^ constant.other.local.plc
//                                   ^ punctuation.definition.variable.plc
//                                           ^ punctuation.separator.sequence.plc
      DSTBLK                      := "DB2".dst
//^^^^^^^^^^^^^^^^^^^^^^^^^^^^^^^^^^^^^^^^^^^^ meta.block.fc.body.plc meta.block.network.plc meta.function-call.arguments.plc meta.group.plc
//    ^^^^^^ variable.parameter.plc
//                                ^^ keyword.operator.assignment.plc
//                                   ^^^^^^^^^ meta.path.plc
//                                   ^^^^^ variable.namespace.plc
//                                   ^ punctuation.definition.variable.begin.plc
//                                       ^ punctuation.definition.variable.end.plc
//                                        ^ punctuation.accessor.dot.plc
//                                         ^^^ variable.other.member.plc
   );
//^^^ meta.block.fc.body.plc meta.block.network.plc
//^^ meta.function-call.arguments.plc meta.group.plc
// ^ punctuation.section.group.end.plc
//  ^ punctuation.terminator.statement.plc
   END_FUNCTION
// ^^^^^^^^^^^^ meta.block.fc.body
// ^^^^^^^^^^^^ keyword.declaration.fc.end
